Staubli VAL3: outputs.pjx

Parameters version=s7.2 stackSize=0 millimeterUnit=true
Data file=outputs.dtx
